(* PLC project Tc2_MC2, Institute of Astronomy OntoManager 0.0.1 *)
(* stored: creationDateTime 2024-08-12T10:53:03.974270, modificationDateTime 2024-08-12T10:53:03.974270 *)

TYPE ST_AxisStatus : STRUCT
  UpdateTaskIndex : BYTE;  (* Task-Index of the task that updated this data set *)
  UpdateCycleTime : LREAL;  (* Task cycle time of the task which calls the status function *)
  CycleCounter : UDINT;  (* PLC cycle counter when this data set updated *)
  NcCycleCounter : LREAL;  (* NC cycle counter incremented after NC task updated NcToPlc data structures *)
  Error : BOOL;  (* Axis error state *)
  ErrorId : UDINT;  (* Axis error code *)
  Disabled : LREAL;  (* Disabled state according to the PLCopen motion control statemachine* ) *)
  ControlLoopClosed : BOOL;  (* Is the control loop closed? *)
  ExtSetPointGenEnabled : BOOL;  (* Is the external setpoint generator enabled? *)
END_STRUCT;
END_TYPE

TYPE PLCTONC_AXIS_REF : STRUCT
  ControlDWord : DWORD;  (* Control double word *)
  Override : DWORD;  (* Velocity override *)
  AxisModeRequest : DWORD;  (* Axis operating mode (PLC request) *)
  AxisModeDWord : DWORD;  (* Optional mode parameter *)
  AxisModeLReal : LREAL;  (* Optional mode parameter *)
  PositionCorrection : LREAL;  (* Correction value for current position *)
  ExtSetPos : LREAL;  (* External position setpoint *)
  ExtSetVelo : LREAL;  (* External velocity setpoint *)
  ExtSetAcc : LREAL;  (* External acceleration setpoint *)
  ExtSetDirection : DINT;  (* External direction setpoint *)
  ExtControllerOutput : LREAL;  (* External controller output *)
  GearRatio1 : LREAL;  (* Gear ratio for dynamic multi master coupling modes *)
  GearRatio2 : LREAL;  (* Gear ratio for dynamic multi master coupling modes *)
  GearRatio3 : LREAL;  (* Gear ratio for dynamic multi master coupling modes *)
  GearRatio4 : LREAL;  (* Gear ratio for dynamic multi master coupling modes *)
END_STRUCT;
END_TYPE

TYPE NCTOPLC_AXIS_REF : STRUCT
  StateDWord : DWORD;  (* Status double word *)
  ErrorCode : DWORD;  (* Axis error code *)
  AxisState : DWORD;  (* Axis moving status *)
  AxisModeConfirmation : DWORD;  (* Axis mode confirmation (feedback from NC) *)
  HomingState : DWORD;  (* State of axis calibration (homing) *)
  CoupleState : DWORD;  (* Axis coupling state *)
  SvbEntries : DWORD;  (* SVB entries/orders (SVB = Set preparation task) *)
  SafEntries : DWORD;  (* SAF entries/orders (SAF = Set execution task) *)
  AxisId : DWORD;  (* Axis ID *)
  OpModeDWord : DWORD;  (* Current operation mode *)
  ActiveControlLoopIndex : WORD;  (* Active control loop index *)
  ControlLoopIndex : WORD;  (* Axis control loop index (0, 1, 2, when multiple control loops are used) *)
  ActPos : LREAL;  (* Actual position (absolut value from NC) *)
  ModuloActPos : LREAL;  (* comment : Actual modulo positio *)
  ModuloActTurns : DINT;  (* Actual modulo turns *)
  ActVelo : LREAL;  (* Actual velocity *)
  PosDiff : LREAL;  (* Position difference (lag distance) *)
  SetPos : LREAL;  (* Setpoint position *)
  SetVelo : LREAL;  (* Setpoint velocity *)
  SetAcc : LREAL;  (* Setpoint acceleration *)
  TargetPos : LREAL;  (* Estimated target position *)
  ModuloSetPos : LREAL;  (* Setpoint modulo position *)
  ModuloSetTurns : DINT;  (* Setpoint modulo turns *)
  CmdNo : WORD;  (* Continuous actual command number *)
  CmdState : WORD;  (* Command state *)
END_STRUCT;
END_TYPE

FUNCTION_BLOCK AXIS_REF
  VAR_INPUT
    PlcToNc : PLCTONC_AXIS_REF;
  END_VAR
  VAR_OUTPUT
    NcToPlc : NCTOPLC_AXIS_REF;
    Status : ST_AxisStatus;
  END_VAR

          
END_FUNCTION_BLOCK
